Universal Robots URScript: 5_move_to_drop_position_one.script

#https://s3-eu-west-1.amazonaws.com/ur-support-site/18383/scriptmanual_en_1.3.pdf
def move_to_drop_position_one():

    popup("Moving to first drop position", title = "Moving to first drop position", blocking = True)

    move_right_p = p[0.55, 0.20, 0, 0, 0, 0]
    move_straight_p = p[0.55, 0, 0, 0, 0, 0]
    height_reposition = p[0, 0, -0.1, 0, 0, 0]
    #move to the right
    movel(pose_add(get_actual_tcp_pose(), move_right_p))
    #move straight
   # movel(pose_add(get_actual_tcp_pose(), move_straight_p))
    #move down for tooling position
    movel(pose_add(get_actual_tcp_pose(), height_reposition))

end
move_to_drop_position_one()
execute_drop_action()
